FUNCTION_BLOCK Draw_box (* Basic FB with empty ECC *)
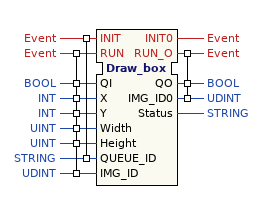
  EVENT_INPUT
    INIT WITH QUEUE_ID;
    RUN WITH X, Y, Width, Height, QI, IMG_ID;
  END_EVENT
  EVENT_OUTPUT
    INIT0;
    RUN_O WITH QO, IMG_ID0;
  END_EVENT
  VAR_INPUT
    QI : BOOL;
    X : INT;
    Y : INT;
    Width : UINT;
    Height : UINT;
    QUEUE_ID : STRING;
    IMG_ID : UDINT;
  END_VAR
  VAR_OUTPUT
    QO : BOOL;
    IMG_ID0 : UDINT;
    Status : STRING;
  END_VAR
END_FUNCTION_BLOCK
